TYPE
  (* Standard: 61499-2; Description: Copyright (c) 2018 fortiss GmbH This program and the accompanying materials are made available under the terms of the Eclipse Public License 2.0 which is available at https://www.eclipse.org/legal/epl-2.0/ SPDX-License-Identifier: EPL-2.0 *)
  (* Version 1.0, 2018-09-26, Jose Cabral, fortiss GmbH *)
  (* ASN.1 tag APPLICATION 1 *)
  PreferredProvider : STRUCT
    providerSystem : ArrowheadSystem;
    providerCloud : ArrowheadCloud;
  END_STRUCT;
END_TYPE
